Fanuc KAREL source: RSET_REALREG.kl

PROGRAM T
%NOLOCKGROUP
VAR
 v0 : STRING[40]
 v1 : BOOLEAN
 v2 : REAL
 v3 : INTEGER
BEGIN
 RSET_REALREG(v0, v1, v2, v3)
END T
